{attribute addProperty BoxType "EL5101-0000-1019"}
{attribute addProperty Id "Latch_C_validAT %I*BOOL811Latch_extern_validAT %I*BOOL812Set_counter_doneAT %I*BOOL813Counter_underflowAT %I*BOOL814Counter_overflowAT %I*BOOL815Status_of_input_statusAT %I*BOOL816Open_circuitAT %I*BOOL817Extrapolation_stallAT %I*BOOL818Status_of_input_AAT %I*BOOL819Status_of_input_BAT %I*BOOL8110Status_of_input_CAT %I*BOOL8111Status_of_input_gateAT %I*BOOL8112Status_of_extern_latchAT %I*BOOL8113Sync_ErrorAT %I*BOOL8132TxPDO_StateAT %I*BOOL817TxPDO_ToggleAT %I*BOOL819Counter_valueAT %I*UINT16217Latch_valueAT %I*UINT16218"}
{attribute addProperty CRC "2786748369"}
{attribute addProperty SizeInBites "160"}
{attribute addProperty SizeInBytes "20"}
TYPE ENC_Status_compact_A61A67D1 :
STRUCT
	{attribute addProperty Name "Latch_C_valid"}
	Latch_C_valid AT %I* : BOOL;
	{attribute addProperty Name "Latch_extern_valid"}
	Latch_extern_valid AT %I* : BOOL;
	{attribute addProperty Name "Set_counter_done"}
	Set_counter_done AT %I* : BOOL;
	{attribute addProperty Name "Counter_underflow"}
	Counter_underflow AT %I* : BOOL;
	{attribute addProperty Name "Counter_overflow"}
	Counter_overflow AT %I* : BOOL;
	{attribute addProperty Name "Status_of_input_status"}
	Status_of_input_status AT %I* : BOOL;
	{attribute addProperty Name "Open_circuit"}
	Open_circuit AT %I* : BOOL;
	{attribute addProperty Name "Extrapolation_stall"}
	Extrapolation_stall AT %I* : BOOL;
	{attribute addProperty Name "Status_of_input_A"}
	Status_of_input_A AT %I* : BOOL;
	{attribute addProperty Name "Status_of_input_B"}
	Status_of_input_B AT %I* : BOOL;
	{attribute addProperty Name "Status_of_input_C"}
	Status_of_input_C AT %I* : BOOL;
	{attribute addProperty Name "Status_of_input_gate"}
	Status_of_input_gate AT %I* : BOOL;
	{attribute addProperty Name "Status_of_extern_latch"}
	Status_of_extern_latch AT %I* : BOOL;
	{attribute addProperty Name "Sync_Error"}
	Sync_Error AT %I* : BOOL;
	{attribute addProperty Name "TxPDO_State"}
	TxPDO_State AT %I* : BOOL;
	{attribute addProperty Name "TxPDO_Toggle"}
	TxPDO_Toggle AT %I* : BOOL;
	{attribute addProperty Name "Counter_value"}
	Counter_value AT %I* : UINT;
	{attribute addProperty Name "Latch_value"}
	Latch_value AT %I* : UINT;
END_STRUCT
END_TYPE

(* stored: Version 1.2.0.0, ProductVersion 3.1.4024.9
   DUT ENC_Status_compact_A61A67D1: Id {fcad5764-08e8-43c1-bb26-d803723d21ca} *)
